{attribute 'qualified_only'}
{attribute 'strict'}
TYPE E_ChooseSampleInstance :
(
	Base,
	Sub1,
	Sub2,
	Sub3
);
END_TYPE

(* stored: Version 1.1.0.1, ProductVersion 3.1.4024.2
   DUT E_ChooseSampleInstance: Id {cd766ce9-8890-439c-a0ea-46d6c145648c} *)
